{attribute 'GeneratedUsingTerminal: AX8108-0100-0102-0102'}
{attribute addProperty BoxType "AX8108-0100-0102-0102"}
{attribute addProperty Id "Ch_A_AxisMain_InputsCh_A_AxisMain_Inputs_BA7CE8DB8Ch_A_AxisMain_OutputsCh_A_AxisMain_Outputs_A99AE12E2Ch_A_Interpolator_OutputsCh_A_Interpolator_Outputs_462A5F1D8Ch_A_PositionControl_InputsCh_A_PositionControl_Inputs_8CB0F55A4"}
{attribute addProperty CRC "3515641622"}
{attribute addProperty Size "22"}
TYPE Ch_A_D18C6F16 :
STRUCT
	{attribute addProperty Name "Ch_A_AxisMain_Inputs"}
	Ch_A_AxisMain_Inputs  : Ch_A_AxisMain_Inputs_BA7CE8DB;
	{attribute addProperty Name "Ch_A_AxisMain_Outputs"}
	Ch_A_AxisMain_Outputs  : Ch_A_AxisMain_Outputs_A99AE12E;
	{attribute addProperty Name "Ch_A_Interpolator_Outputs"}
	Ch_A_Interpolator_Outputs  : Ch_A_Interpolator_Outputs_462A5F1D;
	{attribute addProperty Name "Ch_A_PositionControl_Inputs"}
	Ch_A_PositionControl_Inputs  : Ch_A_PositionControl_Inputs_8CB0F55A;
END_STRUCT
END_TYPE

(* stored: Version 1.2.0.0, ProductVersion 3.1.4024.9
   DUT Ch_A_D18C6F16: Id {5f9ebefe-9b61-467a-91fd-1fb9e5e6bdb3} *)
